{attribute 'linkalways'} 
{attribute 'no_explicit_call' := 'This FB is a CLASS and must be accessed using methods or properties'}
{attribute 'enable_dynamic_creation'}
FUNCTION_BLOCK Node_F_VN_GetPixelFormat EXTENDS VisionNode
VAR
    ipImage : _ITcVnImage;
    stPixelFormat : _TcVnPixelFormat;
    hrPrev : _HRESULT(S_OK);
	hresult : _HRESULT(S_OK);
END_VAR

METHOD PUBLIC  Clone : I_Node
VAR
	pNode : POINTER TO Node_F_VN_GetPixelFormat;
END_VAR
pNode := __NEW(Node_F_VN_GetPixelFormat);
Clone := pNode^;
END_METHOD

METHOD FB_init : BOOL
VAR_INPUT
	bInitRetains : BOOL; // if TRUE, the retain variables are initialized (warm start / cold start)
	bInCopyCode : BOOL;  // if TRUE, the instance afterwards gets moved into the copy code (online change)
END_VAR
AddInput('ipImage', ipImage);
AddInput('hrPrev', hrPrev);
AddOutput('stPixelFormat', stPixelFormat);
AddOutput('hresult',hresult);
END_METHOD

METHOD PROTECTED OnExecute : HRESULT
hresult.Value := F_VN_GetPixelFormat(
    ipImage := ipImage.Value,
	stPixelFormat := stPixelFormat.Value,
	hrPrev:= hrPrev.Value);
END_METHOD

METHOD PUBLIC PreExecutionCheck
VAR_INPUT
	Check : I_PreExecutionChecks;
END_VAR
IF FAILED(hrPrev.Value) THEN
    RETURN;
END_IF

Check.IsTrue(ipImage.IsValid, 'ipImage must contain an image');
END_METHOD

END_FUNCTION_BLOCK

(* stored: Version 1.1.0.1, ProductVersion 3.1.4024.13
   POU Node_F_VN_GetPixelFormat: Id {80bea73c-33d6-0b2a-2fd5-1939cb49c8b1}, SpecialFunc None
   Folder Constructor: Id {4218661d-a1ae-0889-0803-caae0b38ec84}
   Method Clone: Id {b5f1315c-1615-0a60-1504-6caa8b1a9aca}
   Method FB_init: Id {0200acff-3643-0a44-30db-6e214819f783}
   Method OnExecute: Id {d72085f9-3945-0d3c-2291-092097256afc}
   Method PreExecutionCheck: Id {b8b3af61-4109-061a-35a8-eb1cf5843f40} *)
